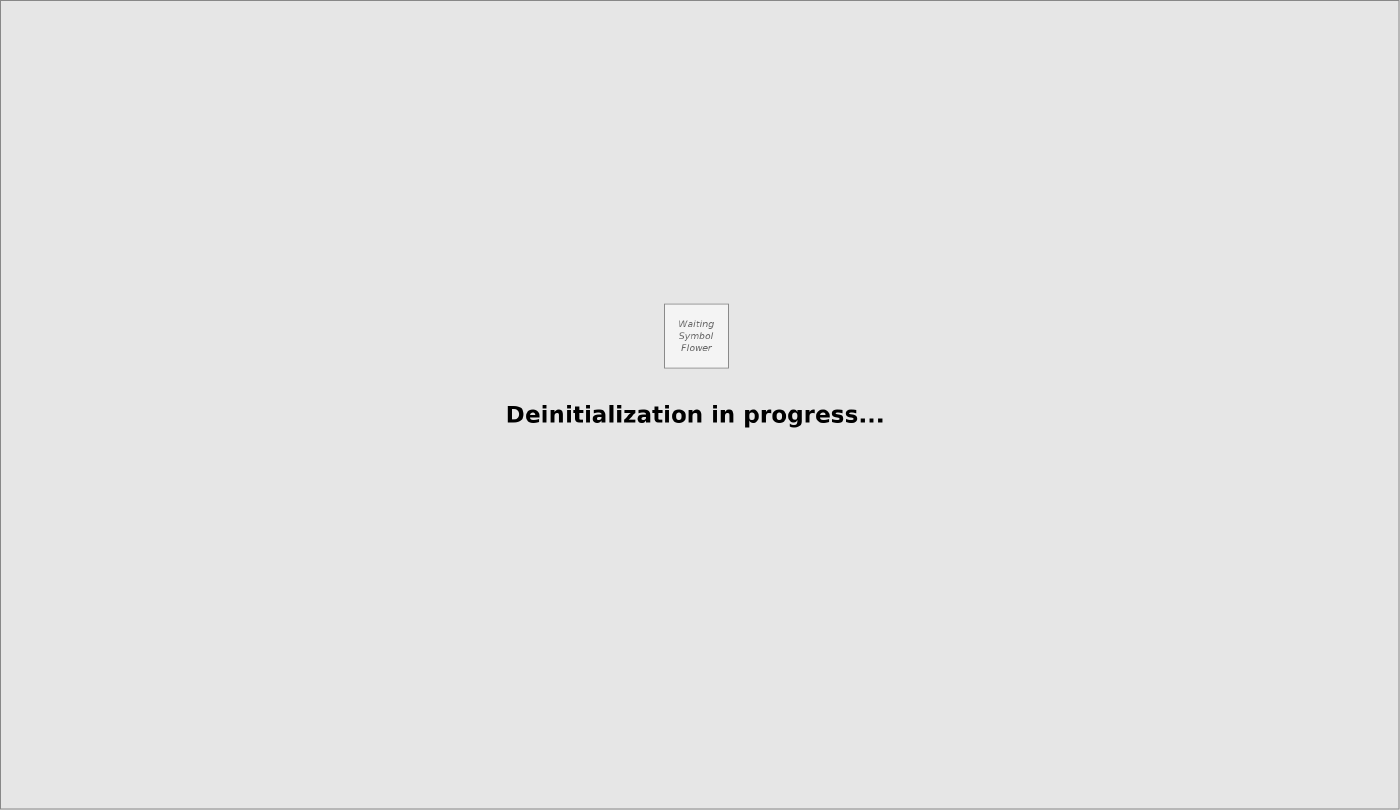
VISUALIZATION PageAborting_1  // 1520x880
    Group (530,330 450x140)
        WaitingSymbolFlower (191,0 70x70)
        Label (0,100 450x40), "Deinitialization in progress..."
END_VISUALIZATION

(* stored: Version 1.1.0.1, ProductVersion 3.1.4024.12
   Visu PageAborting_1: Id {371c2f95-4175-47d6-bb14-7b7f623c1a13} *)
